// SIMATIC S7-200 project (STEP 7-Micro/WIN), CPU 224 CN REL 02.01

SYMBOL_TABLE USER1
Pos_Pieza        I0.0     // Sensor fotoelectrico (presencia de pieza)
Pinza_Cerrada    I0.1     // Sensor indicador de cilindro de dedo Cerrado (pinza)
Cil_Lrg_Ext      I0.2     // Sensor indicador de cilindro largo extendido
Cil_Lrg_Ret      I0.3     // Sensor indicador de cilindro largo retraido
Cil_Del_Ret      I0.4     // Cilindro delgado retraido (hacia arriba)
Cil_Del_Ext      I0.5     // Cilindro delgado extendido (hacia abajo)
Btn_Paro         I1.2     // Pulsador de paro (rojo)
Btn_Marcha       I1.3     // Pulsador de marcha (verde)
Seta_Emerg       I1.4     // Zeta de emergencia
Selector_Rot     I1.5     // Selector rotatorio
V_Pinza          Q0.0     // Valvula del cilindro de dedo (pinza)
V_Cil_Lrg        Q0.2     // Valvula cilindro largo
V_Cil_Del        Q0.3     // Valvula cilindro delgado
Lamp_Amarilla    Q0.7     // Lampara de senalizacion amarilla (falla o advertencia)
Lamp_Verde       Q1.0     // Lampara de senalizacion verde (marcha)
Lamp_Roja        Q1.1     // Lampara de senalizacion roja (paro o falla)
P0_Reposo        M0.0     // Estado de espera inicial
P1_Sujecion      M0.1     // Estado de sujecion de la pieza
P2_Traslacion_In M0.2     // Estado de desplazamiento del carro hacia la prensa
P3_Prensado_Baja M0.3     // Estado de mecanizado (prensa desciende)
P4_Prensado_Sube M0.4     // Estado de retorno de la prensa
P5_Traslacion_Out M0.5     // Estado de retorno del carro
T0_Inicio        M1.0     // Transicion Inicio Ciclo
T1_Sujeto        M1.1     // Transicion Sujecion OK
T2_Carro_Prensa  M1.2     // Transicion Carro en Prensa
T3_Prensa_Abajo  M1.3     // Transicion Prensa Abajo
T4_Prensa_Arriba M1.4     // Transicion Prensa Arriba
T5_Carro_Origen  M1.5     // Transicion Carro en Origen
Ev_Marcha        M2.0     // Evento Marcha presionado y Seta OK
Ev_Pieza         M2.1     // Evento Pieza en recepcion detectada
Ev_Pinza_Cer     M2.2     // Evento Pinza cerrada
Ev_CilL_Ext      M2.3     // Evento Cilindro largo extendido (Origen)
Ev_CilL_Ret      M2.4     // Evento Cilindro largo retraido (Prensa)
Ev_CilD_Ext      M2.5     // Evento Cilindro delgado extendido (Abajo)
Ev_CilD_Ret      M2.6     // Evento Cilindro delgado retraido (Arriba)
Sol_PE           V0.0     // Solicitud Procesamiento a Ensamblaje
Ack_Sol_PE       V1.0     // Reconocimiento PE
Ack_MP           V0.1     // Reconocimiento marcha Unidad de Procesammiento
Marcha_P         V1.1     // Solicitud de marcha para la Unidad de Procesamiento
Proc_OK          V0.2     // Unidad de procesamiento disponible
END_SYMBOL_TABLE

SYMBOL_TABLE S7-200 Symbols
First_Scan_On    SM0.1    // 仅第一个扫描周期中接通为 ON
END_SYMBOL_TABLE

ORGANIZATION_BLOCK MAIN:OB1
TITLE=UNIDAD DE PROCESAMIENTO - RED DE PETRI (CIPN) - 5 MODULOS
//  LOGICA BASADA EN REDES DE PETRI INTERPRETADAS
//  MODULO 1: INICIALIZACION
//  MODULO 2: EVENTOS
//  MODULO 3: DISPARO
//  MODULO 4: DINAMICA
//  MODULO 5: ACCIONES
BEGIN
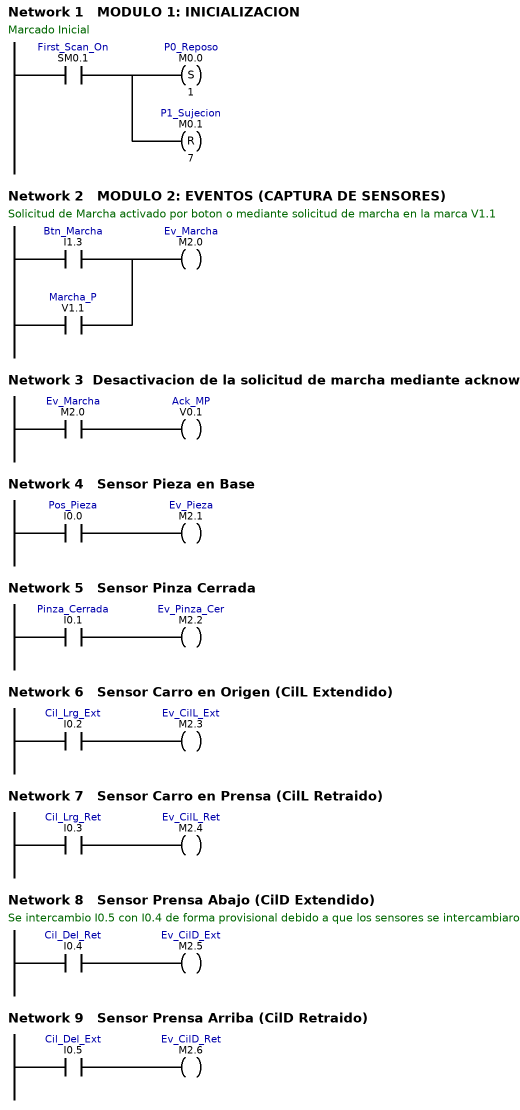
Network 1 //  MODULO 1: INICIALIZACION
//  Marcado Inicial
// P0 Reposo activo
// Limpieza de marcas P1 a M0.7
LD     First_Scan_On:SM0.1
S      P0_Reposo:M0.0, 1
R      P1_Sujecion:M0.1, 7
Network 2 //  MODULO 2: EVENTOS (CAPTURA DE SENSORES)
//  Solicitud de Marcha activado por boton o mediante solicitud de marcha en la marca V1.1
LD     Btn_Marcha:I1.3
O      Marcha_P:V1.1
=      Ev_Marcha:M2.0
Network 3 // Desactivacion de la solicitud de marcha mediante acknowledgement
LD     Ev_Marcha:M2.0
=      Ack_MP:V0.1
Network 4 //  Sensor Pieza en Base
LD     Pos_Pieza:I0.0
=      Ev_Pieza:M2.1
Network 5 //  Sensor Pinza Cerrada
LD     Pinza_Cerrada:I0.1
=      Ev_Pinza_Cer:M2.2
Network 6 //  Sensor Carro en Origen (CilL Extendido)
LD     Cil_Lrg_Ext:I0.2
=      Ev_CilL_Ext:M2.3
Network 7 //  Sensor Carro en Prensa (CilL Retraido)
LD     Cil_Lrg_Ret:I0.3
=      Ev_CilL_Ret:M2.4
Network 8 //  Sensor Prensa Abajo (CilD Extendido)
// Se intercambio I0.5 con I0.4 de forma provisional debido a que los sensores se intercambiaron
LD     Cil_Del_Ret:I0.4
=      Ev_CilD_Ext:M2.5
Network 9 //  Sensor Prensa Arriba (CilD Retraido)
LD     Cil_Del_Ext:I0.5
=      Ev_CilD_Ret:M2.6
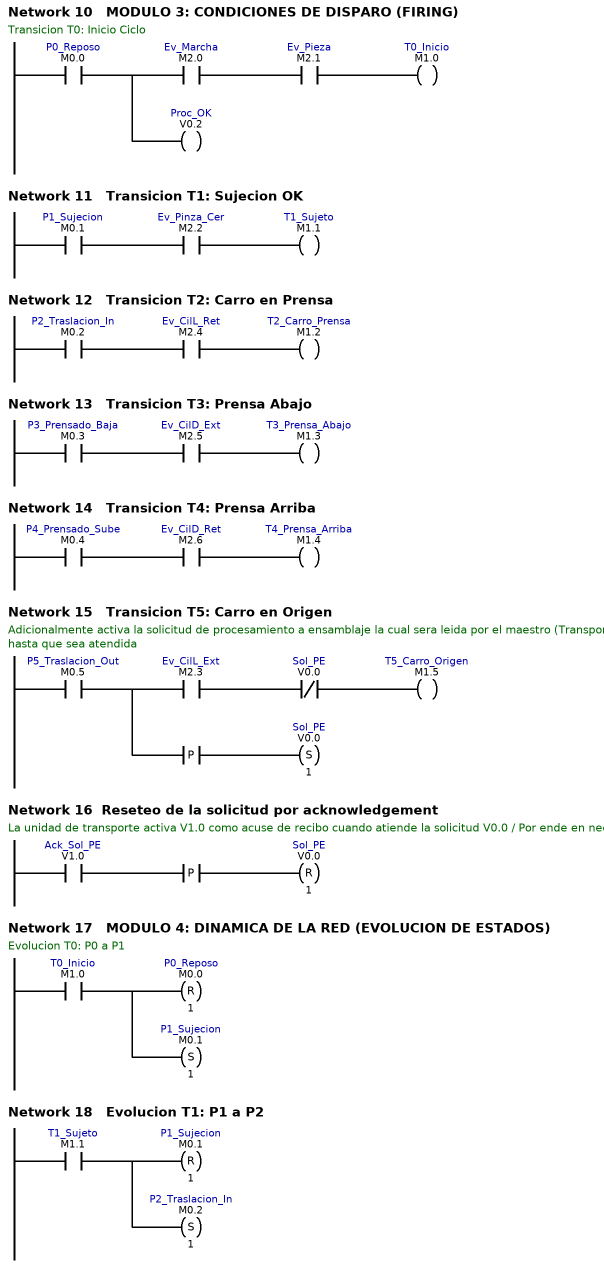
Network 10 //  MODULO 3: CONDICIONES DE DISPARO (FIRING)
//  Transicion T0: Inicio Ciclo
LD     P0_Reposo:M0.0
LPS
A      Ev_Marcha:M2.0
A      Ev_Pieza:M2.1
=      T0_Inicio:M1.0
LPP
=      Proc_OK:V0.2
Network 11 //  Transicion T1: Sujecion OK
LD     P1_Sujecion:M0.1
A      Ev_Pinza_Cer:M2.2
=      T1_Sujeto:M1.1
Network 12 //  Transicion T2: Carro en Prensa
LD     P2_Traslacion_In:M0.2
A      Ev_CilL_Ret:M2.4
=      T2_Carro_Prensa:M1.2
Network 13 //  Transicion T3: Prensa Abajo
LD     P3_Prensado_Baja:M0.3
A      Ev_CilD_Ext:M2.5
=      T3_Prensa_Abajo:M1.3
Network 14 //  Transicion T4: Prensa Arriba
LD     P4_Prensado_Sube:M0.4
A      Ev_CilD_Ret:M2.6
=      T4_Prensa_Arriba:M1.4
Network 15 //  Transicion T5: Carro en Origen
// Adicionalmente activa la solicitud de procesamiento a ensamblaje la cual sera leida por el maestro (Transporte)
// Esta solicitud funciona como enclavamiento que impide volver al estado de reposo hasta que sea atendida
LD     P5_Traslacion_Out:M0.5
LPS
A      Ev_CilL_Ext:M2.3
AN     Sol_PE:V0.0
=      T5_Carro_Origen:M1.5
LPP
EU
S      Sol_PE:V0.0, 1
Network 16 // Reseteo de la solicitud por acknowledgement
// La unidad de transporte activa V1.0 como acuse de recibo cuando atiende la solicitud V0.0
// Por ende en necesario desactivar la solicitud para evitar repeticiones.
LD     Ack_Sol_PE:V1.0
EU
R      Sol_PE:V0.0, 1
Network 17 //  MODULO 4: DINAMICA DE LA RED (EVOLUCION DE ESTADOS)
//  Evolucion T0: P0 a P1
LD     T0_Inicio:M1.0
R      P0_Reposo:M0.0, 1
S      P1_Sujecion:M0.1, 1
Network 18 //  Evolucion T1: P1 a P2
LD     T1_Sujeto:M1.1
R      P1_Sujecion:M0.1, 1
S      P2_Traslacion_In:M0.2, 1
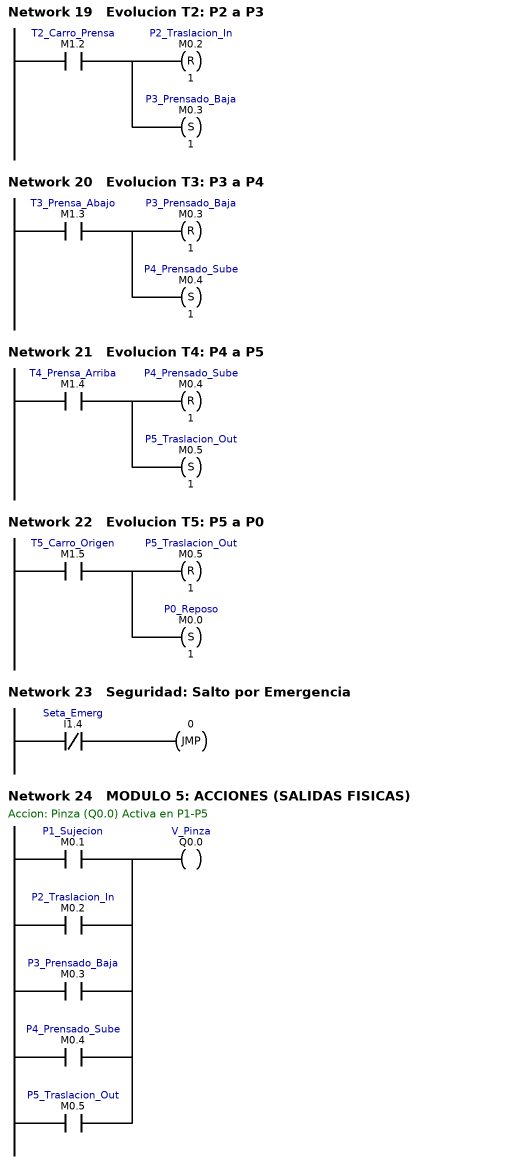
Network 19 //  Evolucion T2: P2 a P3
LD     T2_Carro_Prensa:M1.2
R      P2_Traslacion_In:M0.2, 1
S      P3_Prensado_Baja:M0.3, 1
Network 20 //  Evolucion T3: P3 a P4
LD     T3_Prensa_Abajo:M1.3
R      P3_Prensado_Baja:M0.3, 1
S      P4_Prensado_Sube:M0.4, 1
Network 21 //  Evolucion T4: P4 a P5
LD     T4_Prensa_Arriba:M1.4
R      P4_Prensado_Sube:M0.4, 1
S      P5_Traslacion_Out:M0.5, 1
Network 22 //  Evolucion T5: P5 a P0
LD     T5_Carro_Origen:M1.5
R      P5_Traslacion_Out:M0.5, 1
S      P0_Reposo:M0.0, 1
Network 23 //  Seguridad: Salto por Emergencia
LDN    Seta_Emerg:I1.4
JMP    0
Network 24 //  MODULO 5: ACCIONES (SALIDAS FISICAS)
//  Accion: Pinza (Q0.0) Activa en P1-P5
LD     P1_Sujecion:M0.1
O      P2_Traslacion_In:M0.2
O      P3_Prensado_Baja:M0.3
O      P4_Prensado_Sube:M0.4
O      P5_Traslacion_Out:M0.5
=      V_Pinza:Q0.0
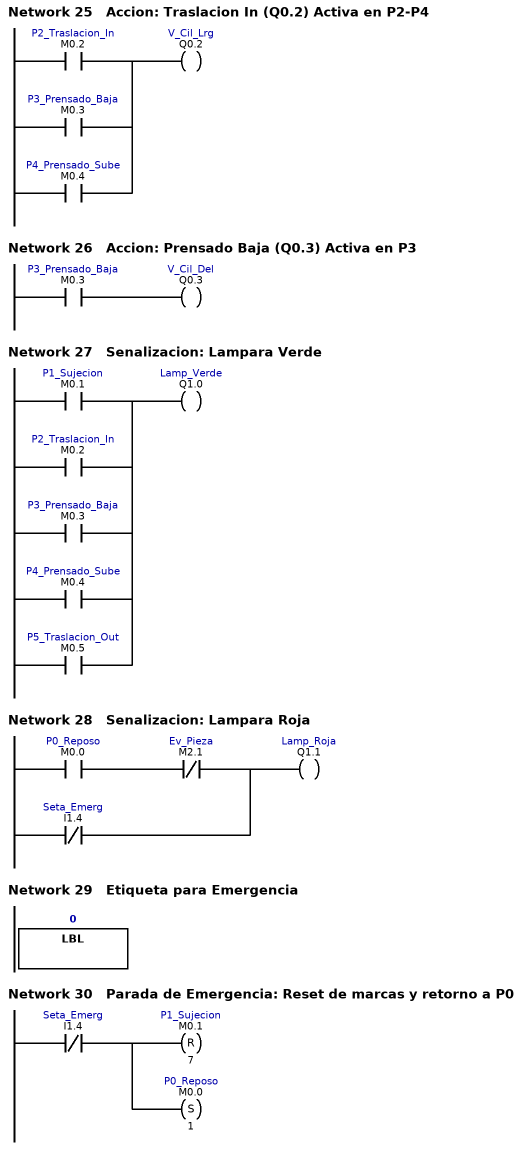
Network 25 //  Accion: Traslacion In (Q0.2) Activa en P2-P4
LD     P2_Traslacion_In:M0.2
O      P3_Prensado_Baja:M0.3
O      P4_Prensado_Sube:M0.4
=      V_Cil_Lrg:Q0.2
Network 26 //  Accion: Prensado Baja (Q0.3) Activa en P3
LD     P3_Prensado_Baja:M0.3
=      V_Cil_Del:Q0.3
Network 27 //  Senalizacion: Lampara Verde
LD     P1_Sujecion:M0.1
O      P2_Traslacion_In:M0.2
O      P3_Prensado_Baja:M0.3
O      P4_Prensado_Sube:M0.4
O      P5_Traslacion_Out:M0.5
=      Lamp_Verde:Q1.0
Network 28 //  Senalizacion: Lampara Roja
LD     P0_Reposo:M0.0
AN     Ev_Pieza:M2.1
ON     Seta_Emerg:I1.4
=      Lamp_Roja:Q1.1
Network 29 //  Etiqueta para Emergencia
LBL    0
Network 30 //  Parada de Emergencia: Reset de marcas y retorno a P0
LDN    Seta_Emerg:I1.4
R      P1_Sujecion:M0.1, 7
S      P0_Reposo:M0.0, 1
END_ORGANIZATION_BLOCK
